// LS Electric XG5000 project: test123
// PLC LSPLC

PROGRAM NewProgram (task: 스캔 프로그램)

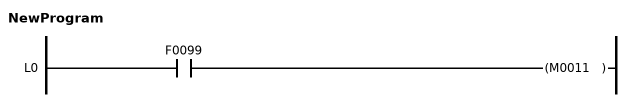
; L0
LOAD      F0099
OUT       M0011